INTERFACE I_Vehicle

METHOD Drive : BOOL
VAR_INPUT
END_VAR
END_METHOD

END_INTERFACE

(* stored: Version 1.1.0.1, ProductVersion 3.1.4024.16
   Itf I_Vehicle: Id {473a2556-85bb-4e54-935a-fa6a9ff19773}
   Method Drive: Id {89500bfd-f906-4133-aa13-91fa3f9818e1} *)
